FUNCTION_BLOCK Tank_Disabled EXTENDS _Tank_State

METHOD OnExecute
IF _ctx.io.in.bEnable THEN
	_ctx.priv.smgr.Request(_ctx.state.iEnabled);
END_IF
END_METHOD

METHOD OnInit
_ctx.io.out.bInletValveOpen := FALSE;
_ctx.hmi.bResetButtonVis := FALSE;
_ctx.priv.IsFillable.Lower();
END_METHOD

END_FUNCTION_BLOCK

(* stored: Version 1.1.0.1
   POU Tank_Disabled: Id {89310616-71c6-4c41-aaa3-c3ff4666422b}, SpecialFunc None
   Method OnExecute: Id {6ce40e97-8db9-4efd-901d-a0bc5d1586ce}
   Method OnInit: Id {252faaa4-8872-40b4-b41b-e23ef6524e6a} *)
